(* CoDeSys 2.3.10.0 project: 2floor.pr6 *)
(* Libraries: STANDARD.LB6 5.6.98 12:03:02 *)

(* Global variable list: Global_Variables *)
VAR_GLOBAL
	din1_1	AT %IX52.0:	BOOL;
	din1_2	AT %IX52.1:	BOOL;
	din1_3	AT %IX52.2:	BOOL;
	din1_4	AT %IX52.3:	BOOL;
	din1_5	AT %IX52.4:	BOOL;
	din1_6	AT %IX52.5:	BOOL;
	din1_7	AT %IX52.6:	BOOL;
	din1_8	AT %IX52.7:	BOOL;
	din2_1	AT %IX53.0:	BOOL;
	din2_2	AT %IX53.1:	BOOL;
	din2_3	AT %IX53.2:	BOOL;
	din2_4	AT %IX53.3:	BOOL;
	din2_5	AT %IX53.4:	BOOL;
	din2_6	AT %IX53.5:	BOOL;
	din2_7	AT %IX53.6:	BOOL;
	din2_8	AT %IX53.7:	BOOL;
	din3_1	AT %IX54.0:	BOOL;
	din3_2	AT %IX54.1:	BOOL;
	din3_3	AT %IX54.2:	BOOL;
	din3_4	AT %IX54.3:	BOOL;
	din3_5	AT %IX54.4:	BOOL;
	din3_6	AT %IX54.5:	BOOL;
	din3_7	AT %IX54.6:	BOOL;
	din3_8	AT %IX54.7:	BOOL;
	din4_1	AT %IX55.0:	BOOL;
	din4_2	AT %IX55.1:	BOOL;
	din4_3	AT %IX55.2:	BOOL;
	din4_4	AT %IX55.3:	BOOL;
	din4_5	AT %IX55.4:	BOOL;
	din4_6	AT %IX55.5:	BOOL;
	din4_7	AT %IX55.6:	BOOL;
	din4_8	AT %IX55.7:	BOOL;
	balkon_peryla	AT %QX52.0:	BOOL;
	dout1_2	AT %QX52.1:	BOOL;
	balkon_bra	AT %QX52.2:	BOOL;
	dout1_4	AT %QX52.3:	BOOL;
	balkon	AT %QX52.4:	BOOL;
	korydor1	AT %QX52.5:	BOOL;
	kino_bra	AT %QX52.6:	BOOL;
	korydor2 AT %QX52.7:	BOOL;
	dout2_1	AT %QX53.0:	BOOL;
	dout2_2	AT %QX53.1:	BOOL;
	dout2_3	AT %QX53.2:	BOOL;
	dout2_4	AT %QX53.3:	BOOL;
	dout2_5	AT %QX53.4:	BOOL;
	dout2_6	AT %QX53.5:	BOOL;
	dout2_7	AT %QX53.6:	BOOL;
	stend	AT %QX53.7:	BOOL;
	dout3_1	AT %QX54.0:	BOOL;
	dout3_2	AT %QX54.1:	BOOL;
	dout3_3	AT %QX54.2:	BOOL;
	dout3_4	AT %QX54.3:	BOOL;
	dout3_5	AT %QX54.4:	BOOL;
	fancoil1_high	AT %QX54.5:	BOOL;
	dout3_7	AT %QX54.6:	BOOL;
	dout3_8	AT %QX54.7:	BOOL;
	dout4_1	AT %QX55.0:	BOOL;
	dout4_2	AT %QX55.1:	BOOL;
	fancoil2_high	AT %QX55.2:	BOOL;
	dout4_4	AT %QX55.3:	BOOL;
	dout4_5	AT %QX55.4:	BOOL;
	dout4_6	AT %QX55.5:	BOOL;
	dout4_7	AT %QX55.6:	BOOL;
	dout4_8	AT %QX55.7:	BOOL;
	skhody	AT %QX56.0:	BOOL;
	dout5_2	AT %QX56.1:	BOOL;
	skhody_peryla	AT %QX56.2:	BOOL;
	dout5_4	AT %QX56.3:	BOOL;
	dout5_5	AT %QX56.4:	BOOL;
	dout5_6	AT %QX56.5:	BOOL;
	dout5_7	AT %QX56.6:	BOOL;
	dout5_8	AT %QX56.7:	BOOL;

	switch16_1: R_TRIG;
	switch13_1: R_TRIG;
	switch14_1: R_TRIG;
	switch14_2: R_TRIG;
	switch15_1: R_TRIG;
	switch15_2: R_TRIG;
	switch15_3: R_TRIG;
	switch17_1: R_TRIG;
	switch17_2: R_TRIG;
	switch18_1: R_TRIG;
	switch18_2: R_TRIG;
	switch18_2_1: R_TRIG;

	switch_kino1: R_TRIG;
	switch_kino2: R_TRIG;
	switch_kino3: R_TRIG;

	switch_trans3: R_TRIG;
	switch_trans1: R_TRIG;
	switch_peryla: R_TRIG;

	peryla1: BOOL;
	peryla3: BOOL;
	peryla2: BOOL;

	timer: TOF;
	timer13_1: TOF;
	timer15_2: TOF;
	timer14_1: TOF;
	timer14_2: TOF;
	timer17_1: TOF;
	timer15_1: TOF;
	timer17_2: TOF;
	timer18_1: TOF;
	timer18_2: TOF;
	timer18_2_1: TOF;
	timer15_3: TOF;
	timer_kino1: TOF;
	timer_kino2: TOF;
	timer_kino3: TOF;
	timer_trans3: TOF;
	timer_trans1: TOF;
	timer_peryla: TOF;
END_VAR

(* POU MAIN, ST *)
PROGRAM MAIN
VAR
END_VAR
triggers;

IF switch15_3.Q AND timer15_3.Q THEN
	stend:=NOT stend;

END_IF;


IF switch15_2.Q AND timer15_2.Q THEN
	dout2_2:=NOT dout2_2;
	dout2_7:=NOT dout2_7;
	peryla2:= NOT peryla2;
END_IF;

IF switch16_1.Q AND timer.Q THEN
	korydor1:=NOT korydor1;
	korydor2:= NOT korydor2;
END_IF;

IF switch17_1.Q AND timer17_1.Q THEN
	dout2_3:=NOT dout2_3;
END_IF;
;

IF switch17_2.Q AND timer17_2.Q THEN
	dout2_1:=NOT dout2_1;
END_IF;

IF switch18_1.Q AND timer18_1.Q THEN
	dout2_6:=NOT dout2_6;
	dout2_4:=NOT dout2_4;
END_IF;

IF switch18_2.Q AND timer18_2.Q THEN
	dout2_5:=NOT dout2_5;
END_IF;

IF switch18_2_1.Q AND timer18_2_1.Q THEN
	dout1_4:=NOT dout1_4;
END_IF;


IF switch_kino1.Q AND timer_kino1.Q THEN
	kino_bra:=NOT kino_bra;
END_IF;

IF switch_kino2.Q AND timer_kino2.Q THEN
	dout1_2:=NOT dout1_2;
END_IF;

IF switch_kino3.Q AND timer_kino3.Q THEN
	balkon_bra:=NOT balkon_bra;
	balkon:=NOT balkon;
	balkon_peryla:= NOT balkon_peryla;
END_IF;

IF switch_trans3.Q AND timer_trans3.Q THEN
	peryla2:= NOT peryla2;
	dout2_2:=NOT dout2_2;
	dout2_7:=NOT dout2_7;
END_IF;

IF switch_trans1.Q AND timer_trans1.Q THEN
	peryla1:= NOT peryla1;
END_IF;

skhody:=din3_7; (*транзит на перший поверх для увімкнення світла на сходах*)
IF switch_peryla.Q AND timer_peryla.Q THEN
	peryla1:= NOT peryla1;
END_IF;

skhody_peryla:=peryla1 OR peryla2;

heat;
END_PROGRAM

(* POU triggers, FBD *)
PROGRAM triggers
VAR





END_VAR
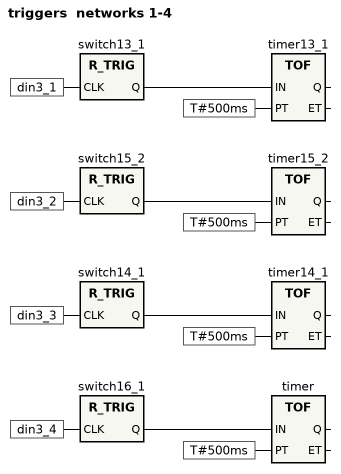
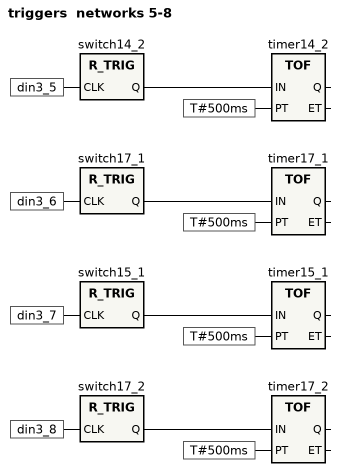
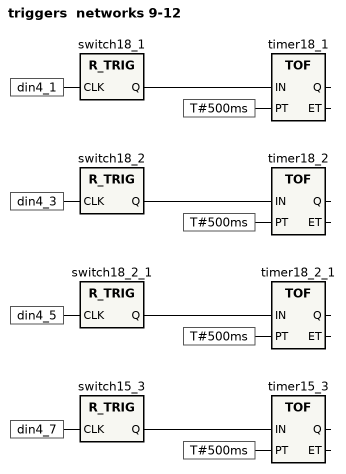
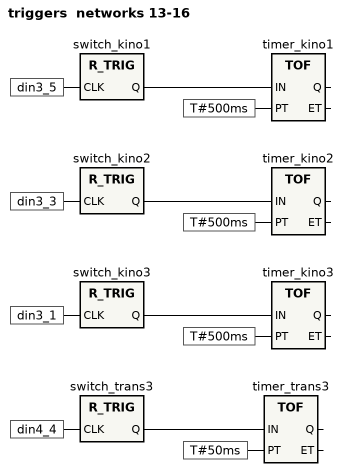
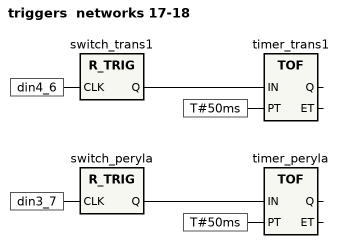
_FBD_ (* Function Block Diagram *)
NETWORK 1
	timer13_1:TOF(IN: switch13_1:R_TRIG(CLK: din3_1), PT: T#500ms)
NETWORK 2
	timer15_2:TOF(IN: switch15_2:R_TRIG(CLK: din3_2), PT: T#500ms)
NETWORK 3
	timer14_1:TOF(IN: switch14_1:R_TRIG(CLK: din3_3), PT: T#500ms)
NETWORK 4
	timer:TOF(IN: switch16_1:R_TRIG(CLK: din3_4), PT: T#500ms)
NETWORK 5
	timer14_2:TOF(IN: switch14_2:R_TRIG(CLK: din3_5), PT: T#500ms)
NETWORK 6
	timer17_1:TOF(IN: switch17_1:R_TRIG(CLK: din3_6), PT: T#500ms)
NETWORK 7
	timer15_1:TOF(IN: switch15_1:R_TRIG(CLK: din3_7), PT: T#500ms)
NETWORK 8
	timer17_2:TOF(IN: switch17_2:R_TRIG(CLK: din3_8), PT: T#500ms)
NETWORK 9
	timer18_1:TOF(IN: switch18_1:R_TRIG(CLK: din4_1), PT: T#500ms)
NETWORK 10
	timer18_2:TOF(IN: switch18_2:R_TRIG(CLK: din4_3), PT: T#500ms)
NETWORK 11
	timer18_2_1:TOF(IN: switch18_2_1:R_TRIG(CLK: din4_5), PT: T#500ms)
NETWORK 12
	timer15_3:TOF(IN: switch15_3:R_TRIG(CLK: din4_7), PT: T#500ms)
NETWORK 13
	timer_kino1:TOF(IN: switch_kino1:R_TRIG(CLK: din3_5), PT: T#500ms)
NETWORK 14
	timer_kino2:TOF(IN: switch_kino2:R_TRIG(CLK: din3_3), PT: T#500ms)
NETWORK 15
	timer_kino3:TOF(IN: switch_kino3:R_TRIG(CLK: din3_1), PT: T#500ms)
NETWORK 16
	timer_trans3:TOF(IN: switch_trans3:R_TRIG(CLK: din4_4), PT: T#50ms)
NETWORK 17
	timer_trans1:TOF(IN: switch_trans1:R_TRIG(CLK: din4_6), PT: T#50ms)
NETWORK 18
	timer_peryla:TOF(IN: switch_peryla:R_TRIG(CLK: din3_7), PT: T#50ms)
_END_FBD_
(* the same logic as Structured Text *)
(* Network 1 *)
switch13_1(CLK := din3_1);
timer13_1(IN := switch13_1.Q, PT := T#500ms);
(* Network 2 *)
switch15_2(CLK := din3_2);
timer15_2(IN := switch15_2.Q, PT := T#500ms);
(* Network 3 *)
switch14_1(CLK := din3_3);
timer14_1(IN := switch14_1.Q, PT := T#500ms);
(* Network 4 *)
switch16_1(CLK := din3_4);
timer(IN := switch16_1.Q, PT := T#500ms);
(* Network 5 *)
switch14_2(CLK := din3_5);
timer14_2(IN := switch14_2.Q, PT := T#500ms);
(* Network 6 *)
switch17_1(CLK := din3_6);
timer17_1(IN := switch17_1.Q, PT := T#500ms);
(* Network 7 *)
switch15_1(CLK := din3_7);
timer15_1(IN := switch15_1.Q, PT := T#500ms);
(* Network 8 *)
switch17_2(CLK := din3_8);
timer17_2(IN := switch17_2.Q, PT := T#500ms);
(* Network 9 *)
switch18_1(CLK := din4_1);
timer18_1(IN := switch18_1.Q, PT := T#500ms);
(* Network 10 *)
switch18_2(CLK := din4_3);
timer18_2(IN := switch18_2.Q, PT := T#500ms);
(* Network 11 *)
switch18_2_1(CLK := din4_5);
timer18_2_1(IN := switch18_2_1.Q, PT := T#500ms);
(* Network 12 *)
switch15_3(CLK := din4_7);
timer15_3(IN := switch15_3.Q, PT := T#500ms);
(* Network 13 *)
switch_kino1(CLK := din3_5);
timer_kino1(IN := switch_kino1.Q, PT := T#500ms);
(* Network 14 *)
switch_kino2(CLK := din3_3);
timer_kino2(IN := switch_kino2.Q, PT := T#500ms);
(* Network 15 *)
switch_kino3(CLK := din3_1);
timer_kino3(IN := switch_kino3.Q, PT := T#500ms);
(* Network 16 *)
switch_trans3(CLK := din4_4);
timer_trans3(IN := switch_trans3.Q, PT := T#50ms);
(* Network 17 *)
switch_trans1(CLK := din4_6);
timer_trans1(IN := switch_trans1.Q, PT := T#50ms);
(* Network 18 *)
switch_peryla(CLK := din3_7);
timer_peryla(IN := switch_peryla.Q, PT := T#50ms);
END_PROGRAM

(* POU heat, ST *)
PROGRAM heat
VAR
END_VAR
{не гріє -32767, гріє - 0
}

Term_32_KL4414_1_Data_Out:=0; {кабінет}
Term_32_KL4414_2_Data_Out:=0; {кінотеатр}
fancoil1_high:=1;
fancoil2_high:=1;
END_PROGRAM
